(* PLC project Unnamed, Unknown Unnamed 1 *)
(* stored: creationDateTime 2023-03-10T10:37:17, modificationDateTime 2023-03-15T15:56:42 *)

(* ISBN 978-3-8348-0266-8, Lernaufgabe 2.4 *)
FUNCTION_BLOCK Reservoirs_Control_System_1
  VAR_INPUT
    IN1 : BOOL;
    IN2 : BOOL;
    IN3 : BOOL;
    IN4 : BOOL;
  END_VAR
  VAR_OUTPUT
    OUTP1 : BOOL;
    OUTP2 : BOOL;
    OUTP3 : BOOL;
    OUTH : BOOL;
  END_VAR
  VAR  (* added by the conversion: wires and edge detectors of the diagram *)
    _OR22_OUT : BOOL;
  END_VAR

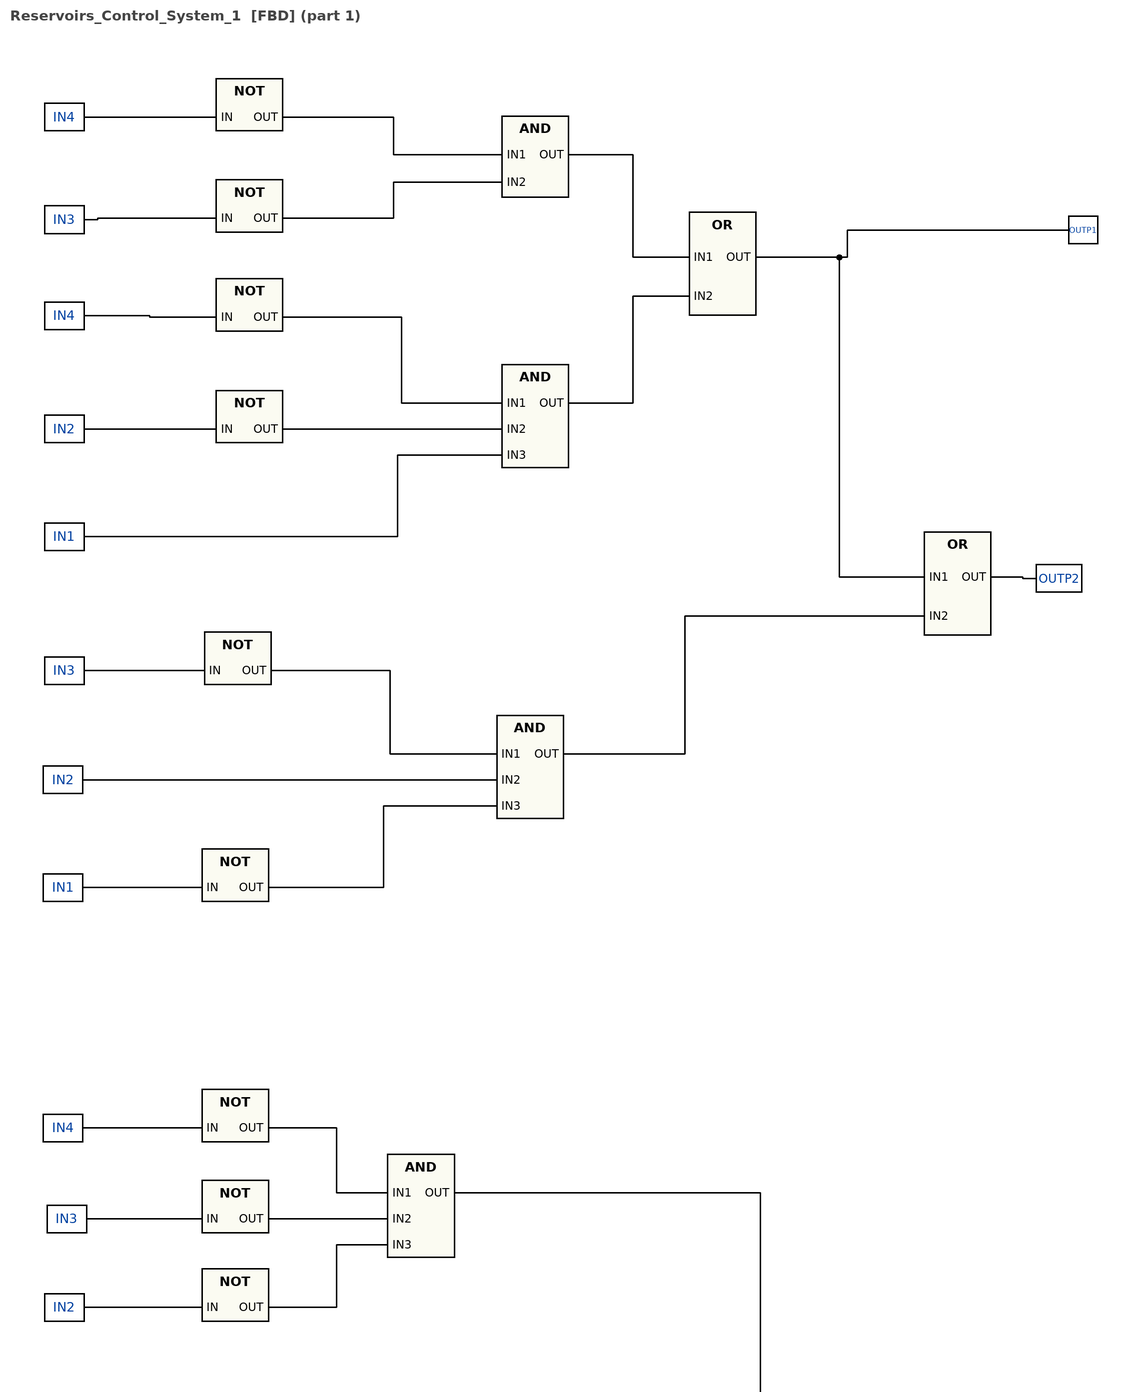
(* FBD diagram, written out as Structured Text *)
_OR22_OUT := NOT IN4 AND NOT IN3 OR NOT IN4 AND NOT IN2 AND IN1;
OUTP1 := _OR22_OUT;
OUTP2 := _OR22_OUT OR NOT IN3 AND IN2 AND NOT IN1;
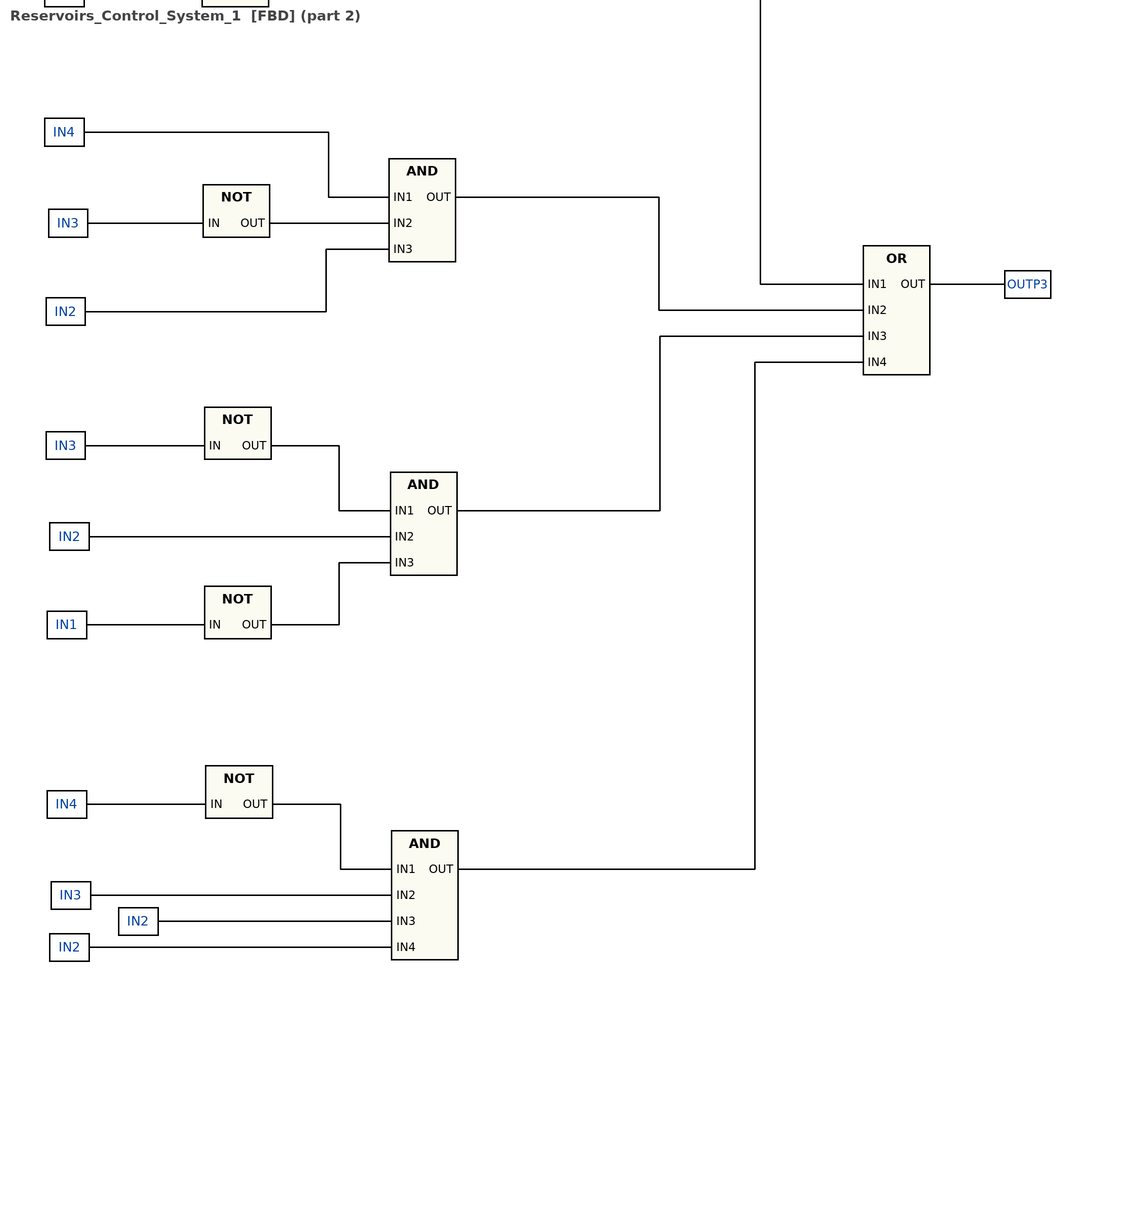
OUTP3 := NOT IN4 AND NOT IN3 AND NOT IN2 OR IN4 AND NOT IN3 AND IN2 OR NOT IN3 AND IN2 AND NOT IN1 OR NOT IN4 AND IN3 AND IN2 AND IN2;
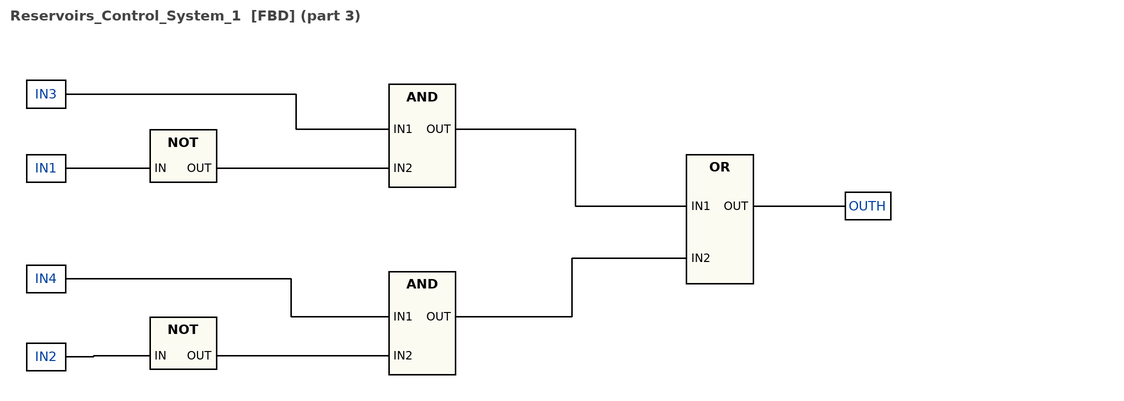
OUTH := IN3 AND NOT IN1 OR IN4 AND NOT IN2;
END_FUNCTION_BLOCK

CONFIGURATION config
  RESOURCE resource1 ON PLC
  END_RESOURCE
END_CONFIGURATION
